// TIA Portal V17 export
// export: Created 2025-08-05T09:36:00.2828713Z, ExportSetting WithDefaults, DisplayName Totally Integrated Automation Portal, DisplayVersion V17, DisplayName TIA Portal Openness, DisplayVersion V17, DisplayName TIA Portal Version Control Interface, DisplayVersion V17, DisplayName SINAMICS Startdrive Advanced, DisplayVersion V17, DisplayName SINAMICS Startdrive G130, G150, S120, S150, SINAMICS MV, S210, DisplayVersion V17, DisplayName SINAMICS Startdrive G110M, G120, G120C, G120D, G120P, G115D, DisplayVersion V17, DisplayName STEP 7 Professional, DisplayVersion V17, DisplayName STEP 7 Safety, DisplayVersion V17, DisplayName WinCC Advanced, DisplayVersion V17
TYPE "typeHmiDataSave"
TITLE = Save HMI data / HMI Daten sichern
// HMI Data backup [V 01.00 | Kernel_V2] / HMI Daten sichern [V 01.00 | Kernel_V2]
// stored: IsFailsafeCompliant false
   STRUCT
      saved : Bool;   // Daten gesichert / Data backed up
      resaved : Bool;   // Daten rückgesichert / Data backed up
      resavedComplete : Bool;   // Daten mit Aktualwerten rückgesichert / Data with actual value backed up
      resavedTrig : Bool;   // Daten rückgesichert Trigger / Data backed up trigger
      saveActive : Bool;   // Daten sichern aktiv / Save data active
      resaveActive : Bool;   // Daten rücksichern aktiv / Backup data active
      resaveCompleteActive : Bool;   // Daten rücksichern mit Aktualwerten aktiv / Backup data with actual values active
      backupBufferInitial : Bool;   // Daten Backup-Puffer ist initial / Data backup buffer initialized
      notUpToDate : Bool;   // Daten Sicherung ist nicht aktuell / Data backup not up to date
   END_STRUCT;
END_TYPE
